FUNCTION WRITE_ANY_TIME_OF_DAY : BOOL
VAR_INPUT
    ptr: POINTER TO TIME_OF_DAY;
    val: TIME_OF_DAY;
END_VAR

ptr^ := val;

END_FUNCTION

(* stored: Version 1.1.0.1, ProductVersion 3.1.4022.9
   POU WRITE_ANY_TIME_OF_DAY: Id {c9020a0a-7555-43c0-b5e9-58aed910df89}, SpecialFunc None *)
